TYPE TAnalogConversion :
STRUCT
	TransducerLoLevel : UINT;
	TransducerHiLevel : UINT;
	ScaledValLoLevel : REAL;
	ScaledValHiLevel : REAL;
END_STRUCT
END_TYPE

(* stored: Version 1.1.0.1, ProductVersion 3.1.4024.13
   DUT TAnalogConversion: Id {d67389dc-2e98-4895-8b46-fbb40c8667e8} *)
